RoboDK station: Nueva Estación (1).rdk

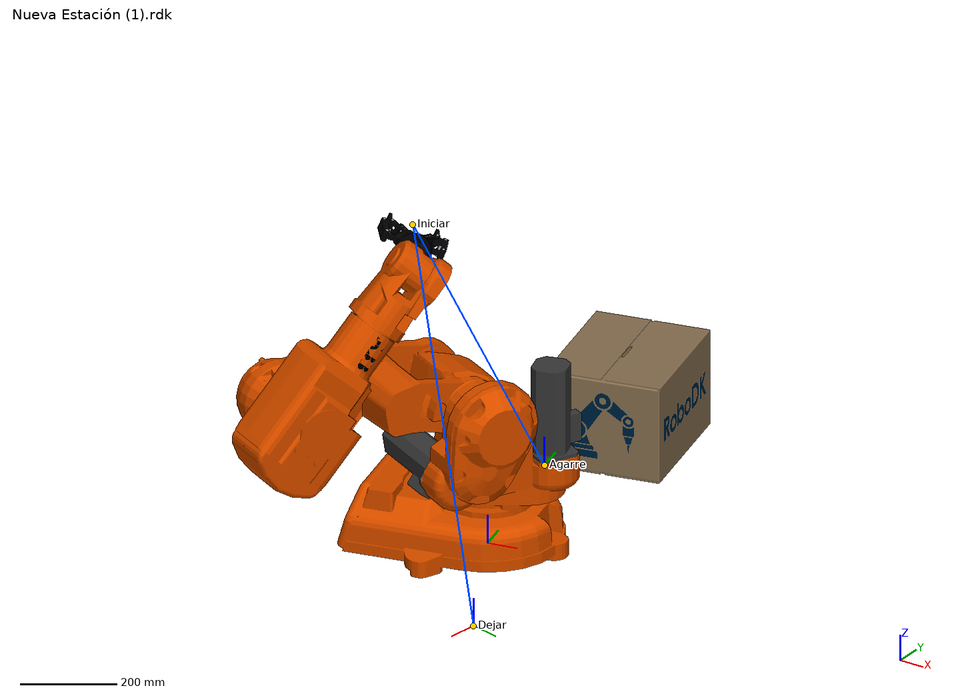
[picture v0: the station drawn from its stored meshes, robots at their saved joint values, targets as dots, program paths as lines]
Station ABB  (saved by RoboDK 5.5.2). Poses are relative to the parent item; angles as X-Y-Z fixed-axis rotations.
  - frame ABB IRB 140-6/0.8 Base at (-61.26, 1858.75, 2122.22) mm, rotated rx 0 ry 0 rz 14.59 deg
    - robot ABB IRB 140-6/0.8: 6 axes, payload 6 kg, reach 810 mm, repeatability 0.03 mm, weight 98 kg
        modified DH rows (alpha deg, a mm, theta deg, d mm): 0, 0, 0, 352; -90, 70, -90, 0; 0, 360, 0, 0; -90, 0, 0, 380; 90, 0, 0, 0; -90, 0, 180, 65
        joint limits [-180, -90, -230, -200, -120, -400] to [180, 110, 50, 200, 120, 400]; home [0, 0, 0, 0, 0, 0]; saved at [-130.942, 85.355, -217.568, -110.315, 69.997, -107.625]
      - tool RobotiQ 2F-85 Gripper (Open), TCP at (0, 0, 140) mm, size 147.4 x 75 x 146.8 mm
  - frame Agarre at (-187.25, 2242.62, 2112.22) mm, rotated rx 0 ry 0 rz 14.6 deg
    - target Iniciar (Cartesian target) at (-161.62, -342.9, 679.61) mm, rotated rx -87.9 ry 21.45 rz 21.68 deg; joints [-70.75, -17.84, -164.77, -200, -4.86, -48.55] of ABB IRB 140-6/0.8
    - target Agarre (Cartesian target) at (0, 0, 0) mm, rotated rx -87.9 ry 21.45 rz 21.68 deg; joints [86.979, 85.918, 2.447, -23.919, -90.463, -67.877] of ABB IRB 140-6/0.8
    - object Box 12x10in (Closed) at (0, 0, 0) mm, size 252 x 305.4 x 216.7 mm, geometry from Box-12x10in-Closed.sld
    - target Dejar (Cartesian target) at (104.36, -699.48, -30) mm, rotated rx -87.9 ry 21.45 rz 21.68 deg; joints [-72.657, 94.452, -16.907, -183.682, -104.387, -69.335] of ABB IRB 140-6/0.8
  - frame Dejar at (90, 1592, 2082.22) mm, rotated rx -1.24 ry 1.51 rz -99.59 deg
  - program Prog1 (9 instructions, listed below)
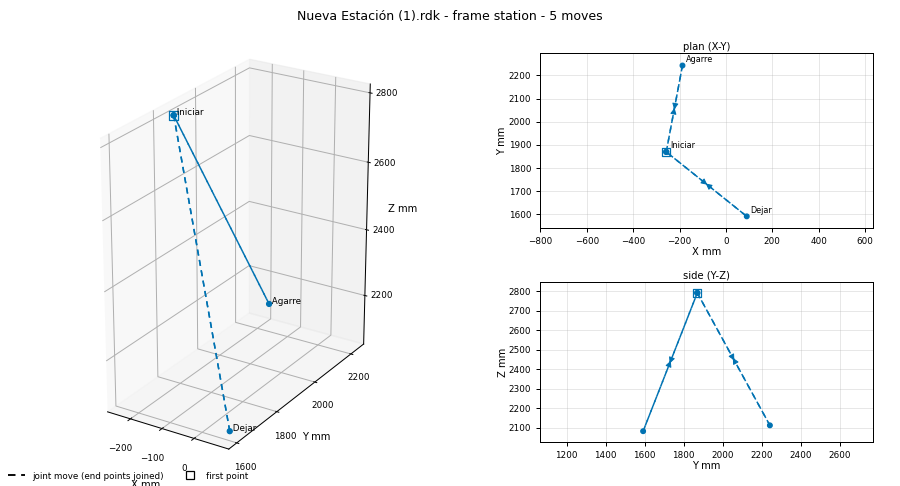
[picture p0: tool path of Nueva Estación (1).rdk in frame station, 5 of 5 moves have a stored position in this frame; points joined in program order, loops and branches not executed]

--- program Prog1 (robot ABB IRB 140-6/0.8) ---
  Est. Ref.: Agarre
  Separar de RobotiQ 2F-85 Gripper (Open)
  MoveJ (Iniciar)
  MoveJ (Agarre)
  Adjuntar a RobotiQ 2F-85 Gripper (Open)
  MoveJ (Iniciar)
  MoveJ (Dejar)
  Separar de RobotiQ 2F-85 Gripper (Open)
  MoveJ (Iniciar)
